TYPE ST_Recipe_Production :
STRUCT
	sName					:STRING[80];
	stInfo					:ST_RecipeInfo;
	stPhase					:ARRAY[0..20] OF ST_Production_Phases;
	iType					:INT; 
	iActivePhase			:INT;
END_STRUCT
END_TYPE

(* stored: Version 1.1.0.1
   DUT ST_Recipe_Production: Id {2f7500cf-31e5-4d11-86f1-a829821fcadd} *)
